	eMBReadInputStatus:
		MBV_Master.ReadInputStatus(
			Quantity								:= wMBVQuantity, 
			MBAddr									:= wMBVAddress, 
			cbLength								:= SIZEOF(wMBVReadData), 
			pMemoryAddr								:= ADR(wMBVReadData), 
			Execute									:= TRUE, 
			Timeout									:= MODBUS_TIMEOUT, 
			BUSY									=> bMBVBusy, 
			Error									=> bMBVError, 
			ErrorId									=> MBV_Errors, 
			cbRead									=> uiMBVRead);
		MBV_Master.ReadInputStatus(BUSY=> bMBVBusy);
		IF NOT MBV_Master.BUSY THEN
			MBV_Master.Execute 						:= FALSE;
			MBV_Master.ReadInputStatus(BUSY=> bMBVBusy);
			IF MBV_Master.Error THEN
				MBV_Master.ReadInputStatus();
			ELSE
				iMBVFunction 						:= 0;			
			END_IF
		END_IF
	
	eMBReadInputRegs:
		MBV_Master.ReadInputRegs(
			Quantity								:= wMBVQuantity, 
			MBAddr									:= wMBVAddress, 
			cbLength								:= SIZEOF(wMBVReadData), 
			pMemoryAddr								:= ADR(wMBVReadData), 
			Execute									:= TRUE, 
			Timeout									:= MODBUS_TIMEOUT, 
			BUSY									=> bMBVBusy, 
			Error									=> bMBVError, 
			ErrorId									=> MBV_Errors, 
			cbRead									=> uiMBVRead);
		MBV_Master.ReadInputRegs(BUSY=> bMBVBusy);
		IF NOT MBV_Master.BUSY THEN
			MBV_Master.Execute 						:= FALSE;
			MBV_Master.ReadInputRegs(BUSY=> bMBVBusy);
			IF MBV_Master.Error THEN
				MBV_Master.ReadInputRegs();
			ELSE
				iMBVFunction 						:= 0;			
			END_IF
		END_IF
	
	eMBWriteSingleCoil:
		MBV_Master.WriteSingleCoil(
			Quantity								:= wMBVQuantity, 
			MBAddr									:= wMBVAddress, 
			cbLength								:= SIZEOF(wMBVWriteData), 
			pMemoryAddr								:= ADR(wMBVWriteData), 
			Execute									:= TRUE, 
			Timeout									:= MODBUS_TIMEOUT, 
			BUSY									=> bMBVBusy, 
			Error									=> bMBVError, 
			ErrorId									=> MBV_Errors, 
			cbRead									=> uiMBVRead);
		MBV_Master.WriteSingleCoil(BUSY=> bMBVBusy);
		IF NOT MBV_Master.BUSY THEN
			MBV_Master.Execute 						:= FALSE;
			MBV_Master.WriteSingleCoil(BUSY=> bMBVBusy);
			IF MBV_Master.Error THEN
				MBV_Master.WriteSingleCoil();
			ELSE
				iMBVFunction 						:= 0;			
			END_IF
		END_IF
	
	eMBWriteMultipleCoils:
		MBV_Master.WriteMultipleCoils(
			Quantity								:= wMBVQuantity, 
			MBAddr									:= wMBVAddress, 
			cbLength								:= SIZEOF(wMBVWriteData), 
			pMemoryAddr								:= ADR(wMBVWriteData), 
			Execute									:= TRUE, 
			Timeout									:= MODBUS_TIMEOUT, 
			BUSY									=> bMBVBusy, 
			Error									=> bMBVError, 
			ErrorId									=> MBV_Errors, 
			cbRead									=> uiMBVRead);
		MBV_Master.WriteMultipleCoils(BUSY=> bMBVBusy);
		IF NOT MBV_Master.BUSY THEN
			MBV_Master.Execute 						:= FALSE;
			MBV_Master.WriteMultipleCoils(BUSY=> bMBVBusy);
			IF MBV_Master.Error THEN
				MBV_Master.WriteMultipleCoils();
			ELSE
				iMBVFunction 						:= 0;			
			END_IF
		END_IF
	
	eMBWriteRegs:
		MBV_Master.WriteRegs(
			Quantity								:= wMBVQuantity, 
			MBAddr									:= wMBVAddress, 
			cbLength								:= SIZEOF(wMBVWriteData), 
			pMemoryAddr								:= ADR(wMBVWriteData), 
			Execute									:= TRUE, 
			Timeout									:= MODBUS_TIMEOUT, 
			BUSY									=> bMBVBusy, 
			Error									=> bMBVError, 
			ErrorId									=> MBV_Errors, 
			cbRead									=> uiMBVRead);
		MBV_Master.WriteRegs(BUSY=> bMBVBusy);
		IF NOT MBV_Master.BUSY THEN
			MBV_Master.Execute 						:= FALSE;
			MBV_Master.WriteRegs(BUSY=> bMBVBusy);
			IF MBV_Master.Error THEN
				MBV_Master.WriteRegs();
			ELSE
				iMBVFunction 						:= 0;			
			END_IF
		END_IF
	
	ELSE
		iMBVFunction 								:= 0;
	
END_CASE
END_ACTION

ACTION A_Status_List:
// Calvin - A_Status_List
// Rev 1.00 - April 23, 2023

strStatusLabel[0] 									:= 'Start Warm Up';
strStatusLabel[1] 									:= 'Warm Up running';
strStatusLabel[2]  									:= 'Start Reactor Reset';
strStatusLabel[3]  									:= 'System ready';
strStatusLabel[4]  									:= 'Evacuation running';
strStatusLabel[5]  									:= 'Steam Bypass running';
strStatusLabel[6]  									:= 'Repressurization running';
strStatusLabel[7]  									:= 'Desorption running';
strStatusLabel[8]  									:= 'Adsorption running';
strStatusLabel[9]  									:= '';
strStatusLabel[10]  								:= 'Stopping process';
strStatusLabel[11]  								:= 'Stopping Warm Up';
strStatusLabel[12]  								:= 'Stopping Evacuation';
strStatusLabel[13]  								:= 'Stopping Steam Bypass';
strStatusLabel[14]  								:= 'Stopping Repressurization';
strStatusLabel[15]  								:= 'Stopping Desorption';
strStatusLabel[16]  								:= 'Stopping Adsorption';
strStatusLabel[17]  								:= '';
strStatusLabel[18]  								:= 'Cycle Error';
strStatusLabel[19]  								:= '';
strStatusLabel[20]  								:= '';
strStatusLabel[21]  								:= 'Fan Test Running';
strStatusLabel[22]  								:= 'Evacuation Error!';
strStatusLabel[23]  								:= 'Steam Bypass Error!';
strStatusLabel[24]  								:= 'Repressurization Error!';
strStatusLabel[25]  								:= 'Desorption Error!';
strStatusLabel[26]  								:= 'Adsorption Error!';
strStatusLabel[27]  								:= '';
strStatusLabel[28]  								:= '';
strStatusLabel[29]  								:= '';
strStatusLabel[30]  								:= 'Evacuation Complete';
strStatusLabel[31]  								:= 'Steam Bypass Complete';
strStatusLabel[32]  								:= 'Repressurization Complete';
strStatusLabel[33]  								:= 'Desoprtion Complete';
strStatusLabel[34]  								:= 'Adsorption Complete';
	
bStatusListLoaded									:= true;
END_ACTION

ACTION A_Temperatures:
// Calvin - A_Temperatures
// Rev 1.00 - June 26, 2023

tgr_TI_1001											:= F_Temperature(TI_1001);
tgb_TI_1001_Error									:= TI_1001_Error;
//bTI_1001_ErrActive									:= SEL(TI_1001_Error, FALSE, bTI_1001_ErrActive);
//gbAlarms[eTC_Alarm]									:= SEL(TI_1001_Error, gbAlarms[eTC_Alarm], TRUE);
                                    				
tgr_TI_1100A										:= F_Temperature(TI_1100A);
tgb_TI_1100A_Error									:= TI_1100A_Error;
//bTI_1100A_ErrActive									:= SEL(TI_1100A_Error, FALSE, bTI_1100A_ErrActive);
//gbAlarms[eTC_Alarm]									:= SEL(TI_1100A_Error, gbAlarms[eTC_Alarm], TRUE);
                                    				
tgr_TI_1100B										:= F_Temperature(TI_1100B);
tgb_TI_1100B_Error									:= TI_1100B_Error;
//bTI_1100B_ErrActive									:= SEL(TI_1100B_Error, FALSE, bTI_1100B_ErrActive);
//gbAlarms[eTC_Alarm]									:= SEL(TI_1100B_Error, gbAlarms[eTC_Alarm], TRUE);

tgr_TI_1100C										:= F_Temperature(TI_1100C);
tgb_TI_1100C_Error									:= TI_1100C_Error;
//bTI_1100C_ErrActive									:= SEL(TI_1100C_Error, FALSE, bTI_1100C_ErrActive);
//gbAlarms[eTC_Alarm]									:= SEL(TI_1100C_Error, gbAlarms[eTC_Alarm], TRUE);
                                    				
tgr_TI_1101											:= F_Temperature(TI_1101);
tgb_TI_1101_Error									:= TI_1101_Error;
//bTI_1101_ErrActive									:= SEL(TI_1101_Error, FALSE, bTI_1101_ErrActive);
//gbAlarms[eTC_Alarm]									:= SEL(TI_1101_Error, gbAlarms[eTC_Alarm], TRUE);
                                    				
tgr_TI_1102A										:= F_Temperature(TI_1102A);
tgb_TI_1102A_Error									:= TI_1102A_Error;
//bTI_1102A_ErrActive									:= SEL(TI_1102A_Error, FALSE, bTI_1102A_ErrActive);
//gbAlarms[eTC_Alarm]									:= SEL(TI_1102A_Error, gbAlarms[eTC_Alarm], TRUE);
                                    				
tgr_TI_1102B										:= F_Temperature(TI_1102B);
tgb_TI_1102B_Error									:= TI_1102B_Error;
//bTI_1102B_ErrActive									:= SEL(TI_1102B_Error, FALSE, bTI_1102B_ErrActive);
//gbAlarms[eTC_Alarm]									:= SEL(TI_1102B_Error, gbAlarms[eTC_Alarm], TRUE);
                                    				
tgr_TI_1103											:= F_Temperature(TI_1103);
tgb_TI_1103_Error									:= TI_1103_Error;
//bTI_1103_ErrActive									:= SEL(TI_1103_Error, FALSE, bTI_1103_ErrActive);
//gbAlarms[eTC_Alarm]									:= SEL(TI_1103_Error, gbAlarms[eTC_Alarm], TRUE);
                                    				
tgr_TI_1104											:= F_Temperature(TI_1104);
tgb_TI_1104_Error									:= TI_1104_Error;
//bTI_1104_ErrActive									:= SEL(TI_1104_Error, FALSE, bTI_1104_ErrActive);
//gbAlarms[eTC_Alarm]									:= SEL(TI_1104_Error, gbAlarms[eTC_Alarm], TRUE);
                                    				
tgr_TI_1105											:= F_Temperature(TI_1105);
tgb_TI_1105_Error									:= TI_1105_Error;
//bTI_1105_ErrActive									:= SEL(TI_1105_Error, FALSE, bTI_1105_ErrActive);
//gbAlarms[eTC_Alarm]									:= SEL(TI_1105_Error, gbAlarms[eTC_Alarm], TRUE);
                                    				
tgr_TI_1106											:= F_Temperature(TI_1106);
tgb_TI_1106_Error									:= TI_1106_Error;
//bTI_1106_ErrActive									:= SEL(TI_1106_Error, FALSE, bTI_1106_ErrActive);
//gbAlarms[eTC_Alarm]									:= SEL(TI_1106_Error, gbAlarms[eTC_Alarm], TRUE);
                                    				
tgr_TI_1301											:= F_Temperature(TI_1301);
tgb_TI_1301_Error									:= TI_1301_Error;
//bTI_1301_ErrActive									:= SEL(TI_1301_Error, FALSE, bTI_1301_ErrActive);
//gbAlarms[eTC_Alarm]									:= SEL(TI_1301_Error, gbAlarms[eTC_Alarm], TRUE);

tgr_TI_1302											:= F_Temperature(TI_1302);
tgb_TI_1302_Error									:= TI_1302_Error;
//bTI_1302_ErrActive									:= SEL(TI_1302_Error, FALSE, bTI_1302_ErrActive);
//gbAlarms[eTC_Alarm]									:= SEL(TI_1302_Error, gbAlarms[eTC_Alarm], TRUE);
                                    	
tgr_TI_1303											:= F_Temperature(TI_1303);
tgb_TI_1303_Error									:= TI_1303_Error;
//bTI_1303_ErrActive									:= SEL(TI_1303_Error, FALSE, bTI_1303_ErrActive);
//gbAlarms[eTC_Alarm]									:= SEL(TI_1303_Error, gbAlarms[eTC_Alarm], TRUE);
                                    				
tgr_TI_1304											:= F_Temperature(TI_1304);
tgb_TI_1304_Error									:= TI_1304_Error;
//bTI_1304_ErrActive									:= SEL(TI_1304_Error, FALSE, bTI_1304_ErrActive);
//gbAlarms[eTC_Alarm]									:= SEL(TI_1304_Error, gbAlarms[eTC_Alarm], TRUE);
                                    	
tgr_TI_1											:= F_Temperature(TI_1);
tgb_TI_1_Error										:= TI_1_Error;

tgr_TI_2											:= F_Temperature(TI_2);
tgb_TI_2_Error										:= TI_2_Error;

tgr_TI_3											:= F_Temperature(TI_3);
tgb_TI_3_Error										:= TI_3_Error;

tgr_TI_4											:= F_Temperature(TI_4);
tgb_TI_4_Error										:= TI_4_Error;

tgr_TI_5											:= F_Temperature(TI_5);
tgb_TI_5_Error										:= TI_5_Error;

tgr_TI_6											:= F_Temperature(TI_6);
tgb_TI_6_Error										:= TI_6_Error;

tgr_TI_7											:= F_Temperature(TI_7);
tgb_TI_7_Error										:= TI_7_Error;

tgr_TI_8											:= F_Temperature(TI_8);
tgb_TI_8_Error										:= TI_8_Error;

tgr_TI_9											:= F_Temperature(TI_9);
tgb_TI_9_Error										:= TI_9_Error;

tgr_TI_10											:= F_Temperature(TI_10);
tgb_TI_10_Error										:= TI_10_Error;

tgr_TI_11											:= F_Temperature(TI_11);
tgb_TI_11_Error										:= TI_11_Error;

tgr_TI_12											:= F_Temperature(TI_12);
tgb_TI_12_Error										:= TI_12_Error;

(*
IF gbAlarms[eTC_Alarm] AND NOT tgb_Active_Alarm THEN
	IF TI_1001_Error AND NOT bTI_1001_ErrActive AND giActiveAlarm = 0 THEN
		bTI_1001_ErrActive							:= TRUE;
		gsTempAlarm									:= '/ TI_1001';
		giActiveAlarm								:= eTC_Alarm;
	ELSIF TI_1100A_Error AND NOT bTI_1100A_ErrActive AND giActiveAlarm = 0 THEN
		bTI_1100A_ErrActive							:= TRUE;
		gsTempAlarm									:= '/ TI_1100A';
		giActiveAlarm								:= eTC_Alarm;
	ELSIF TI_1100B_Error AND NOT bTI_1100B_ErrActive AND giActiveAlarm = 0 THEN
		bTI_1100B_ErrActive							:= TRUE;
		gsTempAlarm									:= '/ TI_1100B';
		giActiveAlarm								:= eTC_Alarm;
	ELSIF TI_1100C_Error AND NOT bTI_1100C_ErrActive AND giActiveAlarm = 0 THEN
		bTI_1100C_ErrActive							:= TRUE;
		gsTempAlarm									:= '/ TI_1100C';
		giActiveAlarm								:= eTC_Alarm;
	ELSIF TI_1101_Error AND NOT bTI_1101_ErrActive AND giActiveAlarm = 0 THEN
		bTI_1101_ErrActive							:= TRUE;
		gsTempAlarm									:= '/ TI_1101';
		giActiveAlarm								:= eTC_Alarm;
	ELSIF TI_1102A_Error AND NOT bTI_1102A_ErrActive AND giActiveAlarm = 0 THEN
		bTI_1102A_ErrActive							:= TRUE;
		gsTempAlarm									:= '/ TI_1102A';
		giActiveAlarm								:= eTC_Alarm;
	ELSIF TI_1102B_Error AND NOT bTI_1102B_ErrActive AND giActiveAlarm = 0 THEN
		bTI_1102B_ErrActive							:= TRUE;
		gsTempAlarm									:= '/ TI_1102B';
		giActiveAlarm								:= eTC_Alarm;
	ELSIF TI_1103_Error AND NOT bTI_1103_ErrActive AND giActiveAlarm = 0 THEN
		bTI_1103_ErrActive							:= TRUE;
		gsTempAlarm									:= '/ TI_1103';
		giActiveAlarm								:= eTC_Alarm;
	ELSIF TI_1104_Error AND NOT bTI_1104_ErrActive AND giActiveAlarm = 0 THEN
		bTI_1104_ErrActive							:= TRUE;
		gsTempAlarm									:= '/ TI_1104';
		giActiveAlarm								:= eTC_Alarm;
	ELSIF TI_1105_Error AND NOT bTI_1105_ErrActive AND giActiveAlarm = 0 THEN
		bTI_1105_ErrActive							:= TRUE;
		gsTempAlarm									:= '/ TI_1105';
		giActiveAlarm								:= eTC_Alarm;
	ELSIF TI_1106_Error AND NOT bTI_1106_ErrActive AND giActiveAlarm = 0 THEN
		bTI_1106_ErrActive							:= TRUE;
		gsTempAlarm									:= '/ TI_1106';
		giActiveAlarm								:= eTC_Alarm;
	ELSIF TI_1301_Error AND NOT bTI_1301_ErrActive AND giActiveAlarm = 0 THEN
		bTI_1301_ErrActive							:= TRUE;
		gsTempAlarm									:= '/ TI_1301';
		giActiveAlarm								:= eTC_Alarm;
	ELSIF TI_1302_Error AND NOT bTI_1302_ErrActive AND giActiveAlarm = 0 THEN
		bTI_1302_ErrActive							:= TRUE;
		gsTempAlarm									:= '/ TI_1302';
		giActiveAlarm								:= eTC_Alarm;
	ELSIF TI_1303_Error AND NOT bTI_1303_ErrActive AND giActiveAlarm = 0 THEN
		bTI_1303_ErrActive							:= TRUE;
		gsTempAlarm									:= '/ TI_1303';
		giActiveAlarm								:= eTC_Alarm;
	ELSIF TI_1304_Error AND NOT bTI_1304_ErrActive AND giActiveAlarm = 0 THEN
		bTI_1304_ErrActive							:= TRUE;
		gsTempAlarm									:= '/ TI_1304';
		giActiveAlarm								:= eTC_Alarm;
	END_IF
END_IF
*)
END_ACTION

ACTION A_WaterHandling:
// Calvin - A_WaterHandling
// Rev 1.00 - September 21, 2023

IF bDrainOn OR tgb_Drains_On THEN
	
	tgb_HS_1200										:= NOT b1200DrainOROff;		//*** Interlock with error
	
	IF tgb_HS_1201_LSH OR (bClearDrains AND tgb_HS_1201_LSL) THEN															// 7/14/23 PS - Adsorption process change
		b1201DrainOn								:= TRUE;
	END_IF
	IF NOT tgb_HS_1201_LSL THEN
		b1201DrainOn								:= FALSE;
	END_IF
	tgb_HS_1201										:= b1201DrainOn AND (tgb_Drains_On OR NOT b1201DrainOROff);

	IF tgb_HS_1202_LSH OR (bClearDrains AND tgb_HS_1202_LSL) THEN															// 7/14/23 PS - Adsorption process change
		b1202DrainOn								:= TRUE;
	END_IF
	IF NOT tgb_HS_1202_LSL THEN
		b1202DrainOn								:= FALSE;
	END_IF
	tgb_HS_1202										:= b1300DrainOn OR b1202DrainOROn OR b1202DrainOn AND (tgb_Drains_On OR NOT b1202DrainOROff);
	tgb_HS_1300B									:= b1300DrainOn;
	
END_IF

rtrigDrainsOff(CLK:= NOT bDrainOn AND NOT tgb_Drains_On);																	// 09/20/23 PS
IF rtrigDrainsOff.Q THEN																									// 09/20/23 PS
	tgb_HS_1200										:= FALSE;
	tgb_HS_1201										:= FALSE;
	tgb_HS_1202										:= FALSE;
	tgb_HS_1300B									:= FALSE;
END_IF

bDrainLSHClear										:= NOT tgb_HS_1202_LSH AND NOT tgb_HS_1201_LSH;
bDrainLSLClear										:= NOT tgb_HS_1202_LSL AND NOT tgb_HS_1201_LSL; 

bCondenserLow										:= tgr_LI_1204 < CONDENSER_LEVEL_LOW_LIMIT;								// 09/19/23 PS
bCondenserFull										:= tgr_LI_1204 > CONDENSER_LEVEL_HIGH_LIMIT;							// 09/21/23 PS
bCondenserRefill									:= tgr_LI_1204 < CONDENSER_LEVEL_REFILL AND NOT bCondenserLow;			// 09/21/23 PS
END_ACTION

ACTION A0_Reset:
// Calvin - A0_Reset
// Rev 1.00 - September 21, 2023

tgr_HS_1102											:= 0;
tgr_IP_1102A										:= 0;
tgr_IP_1102B										:= 0;
tgr_IP_1101											:= 0;
tgr_IP_1302B										:= 0;
tgb_YL_1001											:= FALSE;
tgb_HS_1107											:= FALSE;				
tgb_HS_1101A										:= FALSE;
tgb_HS_1101B										:= FALSE;
tgb_AI_1102A_Pump									:= FALSE;
tgb_AI_1102A_Solenoid								:= FALSE;													
tgb_AI_1102B_Pump									:= FALSE;
tgb_AI_1102B_Solenoid								:= FALSE;													
tgb_HS_1103A										:= FALSE;				
tgb_HS_1103B										:= FALSE;				
tgb_HS_1104											:= FALSE;				
tgb_HS_1203											:= FALSE;				
tgb_HS_1302A										:= FALSE;				
tgb_HS_1301A										:= FALSE;				
tgb_HS_1301											:= FALSE;				
tgb_HS_1301B										:= FALSE;			
tgb_HS_1300A										:= FALSE;			
tgb_HS_1300B										:= FALSE;				
tgb_HS_1305											:= FALSE;
tgb_SV_1201											:= FALSE;
tgb_HT_1_On											:= FALSE;
tgb_HT_2_On											:= FALSE;
tgb_HT_3_On											:= FALSE;
tgb_HT_4_On											:= FALSE;
tgb_HT_5_On											:= FALSE;
tgb_HT_6_On											:= FALSE;
b1201DrainOROff										:= FALSE;
b1202DrainOROff										:= FALSE;
b1202DrainOROn										:= FALSE;
b1300DrainOn										:= FALSE;
bRunValveModulation									:= FALSE;
tgi_Current_Step									:= 0;
strProcessError										:= '';
END_ACTION

ACTION A1_WarmUp:
// Calvin - A1_WarmUp
// Rev 1.00 - September 22, 2023

CASE i1Step OF

	0:	;
	
	1:	
		A0_Reset();
		tgb_AI_1102A_Pump							:= TRUE;
		tgb_AI_1102B_Pump							:= TRUE;
		rTime1										:= VACUUM_TANK_DRAIN_TIME * SECONDS;
		strError									:= gsTK1300HighLevel;
		i1Step										:= i1Step + 1;

	2:	
		bTimer1										:= TRUE;
		IF tgb_HS_1300A_LSH THEN
			b1300DrainOn							:= TRUE;
		ELSE
			bTimer1									:= FALSE;
			b1300DrainOn							:= FALSE;
			IF bCondenserRefill THEN
				rTime2								:= 20 * SECONDS;
				tgb_SV_1201							:= TRUE;
				i1Step								:= i1Step + 1;
			ELSE
				rTime1								:= 10 * MINUTES;
				strError							:= gsBoilerPressureLow;
				i1Step								:= i1Step + 2;
			END_IF
		END_IF
		
	3:
		bTimer2										:= TRUE;
		IF tonTimer2.Q OR bCondenserFull THEN
			bTimer2									:= FALSE;
			tgb_SV_1201								:= FALSE;		
			rTime1									:= 10 * MINUTES;
			strError								:= gsBoilerPressureLow;
			i1Step									:= i1Step + 1;
		END_IF

	4:	
		bTimer1										:= TRUE;
		tgb_YL_1001									:= TRUE;
		IF tgr_PI_1001 > tgr_SP_Boiler_Pressure THEN
			bTimer1									:= FALSE;
			tgb_YL_1001								:= FALSE;
			tgb_Warmup_Complete						:= TRUE;
			i1Step									:= i1Step + 1;
		END_IF

	5:	
		bWarmUpDone									:= TRUE;
		tgi_Current_Step							:= 0;
		i1Step										:= 0;
	
END_CASE

strProcessError										:= SEL(bCondenserLow, strProcessError, gsLowCondenserLevel);					// 09/21/23 PS

IF i1Step > 0 THEN
	IF tonTimer1.Q OR tgb_Stop_Cycle OR strProcessError <> '' THEN
		giActiveAlarm 								:= SEL(tgb_Stop_Cycle, eWarmup_Alarm, eNo_Alarms);
		strError									:= SEL(strProcessError <> '', strError, strProcessError);
		iStep										:= i1Step;		
		A_ClearProcess();
		A0_Reset();
		i1Step										:= 5;
	END_IF
	tgi_Current_Step								:= i1Step;
END_IF
END_ACTION

ACTION A2_Evacuation:
// Calvin - A2_Evacuation
// Rev 1.00 -September 22, 2023

CASE i2Step OF
	
	0:	;
	
	1:	
		A0_Reset();
		tgb_AI_1102A_Pump							:= TRUE;
		tgb_AI_1102B_Pump							:= TRUE;
		gbVacuumHolding								:= FALSE;
		rTime1										:= 30 * SECONDS;
		i2Step										:= 2;
				
	2:	
		IF bDrainLSHClear THEN
			strError								:= gsValvesNotClosed;
			i2Step									:= 4;
		ELSE
			strError								:= gsDrainNotClear;
			i2Step									:= i2Step + 1;
		END_IF
	
	3:	
		bTimer1										:= TRUE;
		IF bDrainLSHClear AND bDrainLSLClear THEN
			bTimer1									:= FALSE;
			strError								:= gsValvesNotClosed;
			i2Step									:= i2Step + 1;
		END_IF

	4:	
		bTimer1										:= TRUE;
		IF gbHS_1102ValvesClosed THEN
			bTimer1									:= FALSE;
			rTime1									:= DEFAULT_STEP_TIME;
			strError								:= gsLRPCoolingFlowLow;
			i2Step									:= i2Step + 1;
		END_IF
	
	5:	
		bTimer1										:= TRUE;
		IF tgb_HS_1300A_LSL AND NOT tgb_HS_1300A_LSH THEN
			tgb_HS_1300A							:= TRUE;
			tgb_HS_1305								:= TRUE;
			tgb_HS_1301								:= TRUE;			
			bTimer1									:= FALSE;
			rTime2									:= 5 * SECONDS;
			i2Step									:= i2Step + 1;
		END_IF
		
	6:	
		bTimer2										:= TRUE;
		IF tonTimer2.Q THEN
			bTimer2									:= FALSE;
			rTime1									:= DEFAULT_STEP_TIME;
			rSP1									:= tgr_SP_Min_LRP_Cooling_Loop_Flow;
			strError								:= gsLRPCoolingFlowLow;
			i2Step									:= i2Step + 1;
		END_IF
	
	7:	
		bTimer1										:= TRUE;
		IF tgr_FI_1300 > rSP1 THEN
			bTimer1									:= FALSE;
			rTime1									:= DEFAULT_STEP_TIME;
			strError								:= gsDrainNotClear;
			i2Step									:= i2Step + 1;
		END_IF			

	8:	
		bTimer1										:= TRUE;
		IF bDrainLSHClear THEN
			b1201DrainOROff							:= TRUE;
			b1202DrainOROff							:= TRUE;
			bTimer1									:= FALSE;
			rTime1									:= DEFAULT_STEP_TIME;
			rSP1									:= tgr_SP_Evacuation_Target_Pressure;
			strError								:= gsTargetPressureHigh;
			i2Step									:= i2Step + 1;
		END_IF
		
	9:	
		bTimer1										:= TRUE;
		IF tgr_PI_1300 < rSP1 THEN
			tgb_HS_1302A							:= TRUE;
			tgb_HS_1107								:= TRUE;
			bTimer1									:= FALSE;
			rTime2									:= 10 * SECONDS;
			i2Step									:= i2Step + 1;
		END_IF

	10:	
		bTimer2										:= TRUE;
		IF tonTimer2.Q THEN
			bTimer2									:= FALSE;
			rTime1									:= DEFAULT_STEP_TIME;
			rSP1									:= tgr_SP_Evacuation_Target_Pressure;
			strError								:= gsTargetPressureHigh;
			i2Step									:= i2Step + 1;
		END_IF
	
	11:	
		bTimer1										:= TRUE;
		IF tgr_PI_1300 <= rSP1 THEN
			bTimer1									:= FALSE;
			tgb_HS_1103A							:= TRUE;
			tgb_HS_1103B							:= TRUE;
			rTime2									:= 10 * SECONDS;
			i2Step									:= i2Step + 1;
		END_IF
		
	12:	
		bTimer2										:= TRUE;
		IF tonTimer2.Q THEN
			bTimer2									:= FALSE;
			rTime1									:= 5 * MINUTES;
			rSP1									:= tgr_SP_Evacuation_Target_Pressure;
			i2Step									:= i2Step + 1;
		END_IF
	
   	13:	
		bTimer1										:= TRUE;
		bInRange1									:= tgr_PI_1300 < rSP1;
		bInRange2									:= tgr_PI_1100 <= rSP1;
		strError									:= SEL(bInRange1, gsPI_1300OutOfRange, gsPI_1100OutOfRange);
		IF bInRange1 AND bInRange2 THEN
			bTimer1									:= FALSE;
			tgb_HS_1103A							:= FALSE;
 	  		tgb_HS_1103B							:= FALSE;
			tgb_HS_1302A							:= FALSE;
			tgb_HS_1301								:= FALSE;
			tgb_HS_1300A							:= FALSE;
			tgb_HS_1305								:= FALSE;
			tgb_HS_1107								:= FALSE;
			rPI_1100_Save							:= tgr_PI_1100;
			rTime2									:= tgr_SP_Leak_Check_Time * SECONDS;
			i2Step									:= i2Step + 1;
		END_IF

	14:	
		bTimer2										:= TRUE;
		IF tonTimer2.Q THEN
			bTimer2									:= FALSE;
			rTime1									:= SECONDS;
			rSP1									:= tgr_SP_Max_Allowed_Pressure_Leakage;
			strError								:= gsVacuumLeak;
			i2Step									:= i2Step + 1;
		END_IF
	
	15:	
		bTimer1										:= TRUE;
		IF ABS(tgr_PI_1100 - rPI_1100_Save) <= rSP1 THEN
			bTimer1									:= FALSE;
			gbVacuumHolding							:= TRUE;
			i2Step									:= i2Step + 1;
		END_IF

	16:	
		b1201DrainOROff								:= FALSE;
		b1202DrainOROff								:= FALSE;
		bEvacuationDone								:= TRUE;
		tgi_Current_Step							:= 0;
		i2Step										:= 0;
		
END_CASE
		
IF i2Step > 0 THEN
	IF tonTimer1.Q OR tgb_Stop_Cycle OR strProcessError <> '' THEN
		giActiveAlarm 								:= SEL(tgb_Stop_Cycle, eEvacuation_Alarm, eNo_Alarms);
		strError									:= SEL(strProcessError <> '', strError, strProcessError);
		iStep										:= i2Step;		
		A_ClearProcess();
		A0_Reset();
		i2Step										:= 16;
	END_IF
	tgi_Current_Step								:= i2Step;
END_IF
END_ACTION

ACTION A3_SteamBypass:
// Calvin - A3_SteamBypass
// Rev 1.00 - September 22, 2023

CASE i3Step OF
	
	0:	;

	1:	
		A0_Reset();
		tgb_AI_1102A_Pump							:= TRUE;
		tgb_AI_1102B_Pump							:= TRUE;
		YL_1001										:= TRUE;
		rTime1										:= VACUUM_TANK_DRAIN_TIME * SECONDS;
		strError									:= gsTK1300HighLevel;
		i3Step										:= i3Step + 1;

	2:	
		bTimer1										:= TRUE;
		IF tgb_HS_1300A_LSH THEN
			b1300DrainOn							:= TRUE;
		ELSE
			bTimer1									:= FALSE;
			b1300DrainOn							:= FALSE;
			IF bCondenserRefill THEN
				rTime2								:= 20 * SECONDS;
				i3Step								:= i3Step + 1;
			ELSE
				rTime1								:= 3 * MINUTES;
				strError							:= gsBoilerPressureLow;
				i3Step								:= i3Step + 2;
			END_IF
		END_IF
		
	3:
		bTimer1										:= TRUE;
		IF NOT bCondenserRefill OR bCondenserFull THEN
			bTimer1									:= FALSE;
			tgb_SV_1201								:= FALSE;		
			tgb_YL_1001								:= TRUE;
			b1201DrainOROff							:= TRUE;
			rTime1									:= 3 * MINUTES;
			i3Step									:= i3Step + 1;
		ELSE
			tgb_SV_1201								:= TRUE;
		END_IF
		
	4:	
		bTimer1										:= TRUE;
		strError									:= SEL(tgr_PI_1101 >= tgr_SP_Evacuation_Target_Pressure_Steam, gsBoilerPressureLow, gsTargetPressureHigh);
		IF tgr_PI_1101 < tgr_SP_Evacuation_Target_Pressure_Steam AND tgr_PI_1001 >= tgr_SP_Boiler_Pressure THEN
			bTimer1									:= FALSE;
			b1202DrainOROn							:= TRUE;
			tgb_HS_1203								:= TRUE;
			tgr_IP_1101								:= 100;
			tgb_HS_1107								:= TRUE;
			rTime2									:= 60 * SECONDS;
			i3Step									:= i3Step + 1;
		END_IF
	
	5:	
		bTimer2										:= TRUE;
		IF tonTimer2.Q THEN
			bTimer2									:= FALSE;
			rTime1									:= 3 * MINUTES;
			strError								:= gsSteamFlowLow;
			i3Step									:= i3Step + 1;
		END_IF
		
	6:	
		bTimer1										:= TRUE;
		IF tgr_FI_1001 > tgr_SP_Min_Bypass_Steam_Flow THEN
			bTimer1									:= FALSE;
			rTime2									:= 30 * SECONDS;
			i3Step									:= i3Step + 1;
		END_IF
		
	7:	
		bTimer2										:= TRUE;
		IF tonTimer2.Q THEN
			bTimer2									:= FALSE;
			rTime1									:= 5 * MINUTES;
			strError								:= gsSteamTempLow;
			i3Step									:= i3Step + 1;
		END_IF
	
	8:	
		bTimer1										:= TRUE;
		strProcessError								:= SEL(tgb_TI_1101_Error, strProcessError, gsTI_1101Error);					// 09/20/23 PS
		IF tgr_TI_1101 > tgr_SP_Min_Bypass_Steam_Temp THEN
			bTimer1									:= FALSE;
			tgr_IP_1101								:= 0;
			tgb_HS_1107								:= FALSE;
			rTime1									:= 10 * MINUTES;
			strError								:= gsLimitSwitchError;
			i3Step									:= i3Step + 1;
		END_IF
		
	9:	
		bTimer1										:= TRUE;
		IF NOT tgb_HS_1202_LSH THEN
			bTimer1									:= FALSE;
			b1202DrainOROff							:= TRUE;
			b1202DrainOROn							:= FALSE;
			tgb_HS_1203								:= FALSE;
			i3Step									:= i3Step + 1;
		END_IF
		
	10:	
		bSteamBypassDone							:= TRUE;
		tgi_Current_Step							:= 0;
		i3Step										:= 0;
		
END_CASE
		
strProcessError										:= SEL(bCondenserLow, strProcessError, gsLowCondenserLevel);					// 09/20/23 PS

IF i3Step > 0 THEN
	IF tonTimer1.Q OR tgb_Stop_Cycle OR strProcessError <> '' THEN
		giActiveAlarm 								:= SEL(tgb_Stop_Cycle, eSteamBypass_Alarm, eNo_Alarms);
		strError									:= SEL(strProcessError <> '', strError, strProcessError);		
		iStep										:= i3Step;		
		A_ClearProcess();
		A0_Reset();
		i3Step										:= 10;
	END_IF
	tgi_Current_Step								:= i3Step;
END_IF
END_ACTION

ACTION A4_Desorption:
// Calvin - A4_Desorption
// Rev 1.00 - September 22, 2023

CASE i4Step OF
	
	0:	bOverTemp									:= FALSE;
		
	1:	
		A0_Reset();
		YL_1001										:= TRUE;
		b1201DrainOROff								:= TRUE;
		b1202DrainOROff								:= TRUE;
		rTime1										:= 2 * SECONDS;
		rSP1										:= tgr_SP_Evacuation_Target_Pressure_Steam;								// 07/14/23 PS - Added set point
		strError									:= gsTargetPressureHigh;
		i4Step										:= 2;
	
	2:	
		bTimer1										:= TRUE;
		IF tgr_PI_1100 < rSP1 THEN
			bTimer1									:= FALSE;
			i4Step									:= i4Step + 1;
		END_IF
		
	3:	
		IF gbVacuumHolding THEN
			rTime1									:= DEFAULT_STEP_TIME;
			rSP1									:= tgr_SP_Evacuation_Target_Pressure_Steam;								// 07/14/23 PS - Added set point
			rSP2									:= tgr_SP_Boiler_Pressure;
			i4Step									:= 6;
		ELSE
			rTime2									:= tgr_SP_Leak_Check_Time * SECONDS;
			i4Step									:= i4Step + 1;
		END_IF
		
	4:	
		bTimer2										:= TRUE;
		IF tonTimer2.Q THEN
			bTimer2									:= FALSE;
			rTime1									:= 1 * SECONDS;
			rSP1									:= tgr_SP_Max_Allowed_Pressure_Leakage;
			strError								:= gsVacuumLeak;
			i4Step									:= i4Step + 1;
		END_IF

	5:	
		bTimer1										:= TRUE;
		IF ABS(tgr_PI_1100 - rPI_1100_Save) <= rSP1 THEN
			bTimer1									:= FALSE;
			gbVacuumHolding							:= TRUE;
			rTime1									:= 10 * MINUTES;
			rSP1									:= tgr_SP_Evacuation_Target_Pressure_Steam;								// 07/14/23 PS - Added set point
			rSP2									:= tgr_SP_Boiler_Pressure;
			i4Step									:= i4Step + 1;
		END_IF

	6:	
		bTimer1										:= TRUE;
		bInRange1									:= tgr_PI_1100 < rSP1;
		bInRange2									:= tgr_PI_1001 >= rSP2;
		strError									:= SEL(bInRange1, gsTargetPressureHigh, gsBoilerPressureLow);
		IF bInRange1 AND bInRange2 THEN
			bTimer1									:= FALSE;
			rTime2									:= 5 * SECONDS;
			i4Step									:= i4Step + 1;
		END_IF
		
	7:	
		bTimer2										:= TRUE;
		tgr_IP_1101									:= tgr_SP_Steam_Valve_Percent_Open;
		IF tonTimer2.Q THEN
			bTimer2									:= FALSE;
			rTime1									:= DEFAULT_STEP_TIME;
			strError								:= gsValveOutOfRange;
			i4Step									:= i4Step + 1;
		END_IF
		
	8:	
		bTimer1										:= TRUE;
		bInRange1									:= ABS(tgr_ZT_1101 - tgr_IP_1101) <= 5;
 		IF bInRange1 THEN
			bTimer1									:= FALSE;
			tgb_HS_1101A							:= TRUE;
			tgb_HS_1101B							:= TRUE;
			rTime1									:= 10 * MINUTES;
			strError								:= gsReactorPressureLow;
			i4Step									:= i4Step + 1;
		END_IF

	9:	
		bTimer1										:= TRUE;
		IF tgr_PI_1100 > 0.5 THEN
			bTimer1									:= FALSE;
			gbVacuumHolding							:= FALSE;
			b1201DrainOROff							:= FALSE;
			b1202DrainOROff							:= FALSE;
			rTime1									:= 30 * MINUTES;
			rSP1									:= tgr_SP_Steam_Repressurization_Pressure;
			i4Step									:= i4Step + 1;
		END_IF

	10:	
		bTimer1										:= TRUE;	
		bInRange1									:= tgr_PI_1001 > rSP1;
		bInRange2									:= tgr_PI_1101 > rSP1;
		bInRange3									:= tgr_PI_1100 > rSP1;
		strError									:= SEL(bInRange1, gsPI_1001PressureLow, SEL(bInRange2, gsPI_1101PressureLow, gsPI_1100PressureLow));
		IF bInRange1 AND bInRange2 AND bInRange3 THEN
			bTimer1									:= FALSE;
			tgb_HS_1203								:= TRUE;
			tgb_HS_1300A							:= TRUE;
			tgb_HS_1305								:= TRUE;
			tgb_HS_1301								:= TRUE;
			rTime2									:= 5 * SECONDS;
			i4Step									:= i4Step + 1;
		END_IF
		
	11:	
		bTimer2										:= TRUE;
		IF tonTimer2.Q THEN
			bTimer2									:= FALSE;
			rTime1									:= 20 * SECONDS;
			rSP1									:= tgr_SP_Min_LRP_Cooling_Loop_Flow;
			rSP2									:= tgr_SP_Evacuation_Target_Pressure;
			i4Step									:= i4Step + 1;
		END_IF
	
	12:	
		bTimer1										:= TRUE;
		bInRange1									:= tgr_FI_1300 > rSP1;
		bInRange2									:= tgr_PI_1300 < rSP2;
		IF bInRange1 AND bInRange2 THEN
			bTimer1									:= FALSE;
			tgb_HS_1302A							:= TRUE;
			rTime2									:= 6 * SECONDS;
			i4Step									:= i4Step + 1;
		END_IF
		
	13:	
		bTimer2										:= TRUE;
		IF tonTimer2.Q THEN
			bTimer2									:= FALSE;
			rSP1									:= tgr_SP_Evacuation_Target_Pressure;
			i4Step									:= i4Step + 1;
		END_IF

	14:	
		IF tgr_PI_1300 < rSP1 THEN
			tgr_IP_1302B							:= tgr_SP_IP_1302B_Valve_Low;
		END_IF
		rTime2										:= 3 * SECONDS;
		i4Step										:= i4Step + 1;
		
	15:	
		bTimer2										:= TRUE;
		IF tonTimer2.Q THEN
			bTimer2									:= FALSE;
			rSP1									:= tgr_SP_Evacuation_Target_Pressure;
			strError								:= gsTargetPressureHigh;
			i4Step									:= i4Step + 1;
		END_IF

	16:	
		bTimer1										:= TRUE;
		IF tgr_PI_1300 < rSP1 THEN
			bTimer1									:= FALSE;
			tgb_HS_1103A							:= TRUE;
			tgb_HS_1103B							:= TRUE;
			bRunValveModulation						:= TRUE;
			rTime1									:= 5 * MINUTES;
			rTime2									:= tgr_SP_Steam_Purge_Time * MINUTES;
			strError								:= gsValveOutOfRange;
			i4Step									:= i4Step + 1;
		END_IF
		
	17:	
		bTimer1										:= TRUE;
		bTimer2										:= TRUE;
		IF bValveInRange THEN
			bTimer1									:= FALSE;
			rTime1									:= SECONDS;
			strError								:= gsThermocoupleError;
			i4Step									:= i4Step + 1;
		END_IF
		
	18:	
		bTimer1										:= TRUE;
		IF NOT tgb_TI_1100A_Error OR NOT tgb_TI_1100B_Error OR NOT tgb_TI_1100C_Error THEN
			bTimer1									:= FALSE;
			rSP1									:= tgr_SP_Max_Allowed_Sorbent_Temp;
			rSP2									:= tgr_SP_Steam_Purge_Cutoff_Temp;
			i4Step									:= i4Step + 1;
		END_IF
	
	19:	
		bInRange1									:= NOT tgb_TI_1100A_Error AND tgr_TI_1100A > rSP1;
		bInRange2									:= NOT tgb_TI_1100B_Error AND tgr_TI_1100B > rSP1;
		bInRange3									:= NOT tgb_TI_1100C_Error AND tgr_TI_1100C > rSP1;
		IF bInRange1 OR bInRange2 OR bInRange3 THEN
			bOverTemp								:= TRUE;
			bTimer2									:= FALSE;
			rTime1									:= SECONDS;
			i4Step									:= i4Step + 1;
		ELSE
			bInRange1								:= (NOT tgb_TI_1100A_Error AND tgr_TI_1100A > rSP2) OR tgb_TI_1100A_Error;
			bInRange2								:= (NOT tgb_TI_1100B_Error AND tgr_TI_1100B > rSP2) OR tgb_TI_1100B_Error;
			bInRange3								:= (NOT tgb_TI_1100C_Error AND tgr_TI_1100C > rSP2) OR tgb_TI_1100C_Error;
			IF tonTimer2.Q THEN
				bTimer2								:= FALSE;
				IF bInRange1 AND bInRange2 AND bInRange3 THEN
					i4Step							:= i4Step + 1;
				ELSE
					strProcessError					:= SEL(bOverTemp, gsTempOutOfRange, gsSorbentOverTemp);
				END_IF
			END_IF
		END_IF
		
	20:	
		bRunValveModulation							:= FALSE;
		tgr_IP_1101									:= 0;
		tgr_IP_1302B								:= 0;
		tgb_HS_1101A								:= FALSE;							
		tgb_HS_1101B								:= FALSE;							
		rTime1										:= 5 * MINUTES;
		rSP1										:= 0.5;
		strError									:= gsPI_1100OutOfRange;
		i4Step										:= i4Step + 1;	

	21: 
		bTimer1										:= TRUE;
		IF tgr_PI_1100 < rSP1 THEN
			bTimer1									:= FALSE;
			b1201DrainOROff							:= TRUE;
			b1202DrainOROff							:= TRUE;
			rSP1									:= tgr_SP_Evap_Cooling_Cutoff_Temp;
			rSP2									:= tgr_SP_Evap_Cooling_Target_Pressure;
			rTime1									:= 20 * MINUTES;
			i4Step									:= i4Step + 1;
		END_IF
		
	22:	
		bTimer1										:= TRUE;
		bInRange1									:= (NOT tgb_TI_1100A_Error AND tgr_TI_1100A < rSP1) OR tgb_TI_1100A_Error;
		bInRange2									:= (NOT tgb_TI_1100B_Error AND tgr_TI_1100B < rSP1) OR tgb_TI_1100B_Error;
		bInRange3									:= (NOT tgb_TI_1100C_Error AND tgr_TI_1100C < rSP1) OR tgb_TI_1100C_Error;
		strError									:= SEL(tgr_PI_1100 >= rSP2, gsTempOutOfRange, gsPI_1100OutOfRange);
		IF bInRange1 AND bInRange2 AND bInRange3 AND tgr_PI_1100 < rSP2 THEN
			bTimer1									:= FALSE;
			i4Step									:= i4Step + 1;
		END_IF	
		
	23:	
		tgb_HS_1103A								:= FALSE;
		tgb_HS_1103B								:= FALSE;
		tgb_HS_1302A								:= FALSE;
		tgb_HS_1301									:= FALSE;
		tgb_HS_1305									:= FALSE;
		tgb_HS_1300A								:= FALSE;
		tgb_HS_1203									:= FALSE;
		i4Step										:= i4Step + 1;
		
	24:
		bDesorptionDone								:= TRUE;
		tgi_Current_Step							:= 0;
		i4Step										:= 0;		
	
END_CASE

strProcessError										:= SEL(bCondenserLow, strProcessError, gsLowCondenserLevel);					// 09/07/23 PS

IF i4Step > 0 THEN
	IF tonTimer1.Q OR tgb_Stop_Cycle OR strProcessError <> '' THEN
		giActiveAlarm 								:= SEL(tgb_Stop_Cycle, eDesorption_Alarm, eNo_Alarms);
		strError									:= SEL(strProcessError <> '', strError, strProcessError);		
		iStep										:= i4Step;		
		A_ClearProcess();
		A0_Reset();
		i4Step										:= 24;
	END_IF
	tgi_Current_Step								:= i4Step;
END_IF
END_ACTION

ACTION A5_Repressurization:
// Calvin - A5_Repressurization
// Rev 1.00 - September 22, 2023

CASE i5Step OF
	
	0:	;
		
	1:	
		A0_Reset();
		tgb_AI_1102A_Pump							:= TRUE;
		tgb_AI_1102B_Pump							:= TRUE;
		rTime1										:= SECONDS;
		strError									:= gsThermocoupleError;
		i5Step										:= 2;
		
	2:	
		bTimer1										:= TRUE;
		bTempAGood									:= NOT tgb_TI_1100A_Error;
		bTempBGood									:= NOT tgb_TI_1100B_Error;
		bTempCGood									:= NOT tgb_TI_1100C_Error;
		IF bTempAGood OR bTempBGood OR bTempCGood THEN
			bTimer1									:= FALSE;
			rTime1									:= DEFAULT_STEP_TIME;
			rSP1									:= tgr_SP_Adsorption_Temp;
			strError								:= gsTempOutOfRange;
			i5Step									:= i5Step + 1;
		END_IF
	
	3:	
		bTimer1										:= TRUE;
		bInRange1									:= (bTempAGood AND tgr_TI_1100A < rSP1) OR NOT bTempAGood;
		bInRange2									:= (bTempBGood AND tgr_TI_1100B < rSP1) OR NOT bTempBGood;
		bInRange3									:= (bTempCGood AND tgr_TI_1100C < rSP1) OR NOT bTempCGood;
		IF bInRange1 AND bInRange2 AND bInRange3 THEN
			bTimer1									:= FALSE;
			tgb_HS_1104								:= TRUE;
			rTime1									:= DEFAULT_STEP_TIME;
			rSP1									:= tgr_SP_Reactor_Repressurization_Pressure;
			strError								:= gsPI_1100OutOfRange;			
			i5Step									:= i5Step + 1;
		END_IF
		
	4:	
		bTimer1										:= TRUE;
		IF tgr_PI_1100 > rSP1 THEN
			bTimer1									:= FALSE;
			rTime2									:= 5 * SECONDS;
			i5Step									:= i5Step + 1;			
		END_IF
		
	5:	
		bTimer2										:= TRUE;
		IF tonTimer2.Q THEN
			bTimer2									:= FALSE;
			i5Step									:= i5Step + 1;
		END_IF
		
	6:	
		tgb_HS_1104									:= FALSE;
		i5Step										:= i5Step + 1;
	
	7:	
		bRepressurizationDone						:= TRUE;
		tgi_Current_Step							:= 0;
		i5Step										:= 0;
	
END_CASE

IF i5Step > 0 THEN
	IF tonTimer1.Q OR tgb_Stop_Cycle OR strProcessError <> '' THEN
		giActiveAlarm 								:= SEL(tgb_Stop_Cycle, eRepressurization_Alarm, eNo_Alarms);
		strError									:= SEL(strProcessError <> '', strError, strProcessError);		
		iStep										:= i5Step;		
		A_ClearProcess();
		A0_Reset();
		i5Step										:= 7;
	END_IF
	tgi_Current_Step								:= i5Step;
END_IF
END_ACTION

ACTION A6_Adsorption:
// Calvin - A6_Adsorption
// Rev 1.00 - September 22, 2023

CASE i6Step OF
	
	0:	;
		
	1:	
		A0_Reset();
		tgb_AI_1102A_Pump							:= TRUE;
		tgb_AI_1102B_Pump							:= TRUE;
		bClearDrains								:= FALSE;
		rSP1										:= tgr_SP_Reactor_Repressurization_Pressure;
		strError									:= gsReactorPressureLow;
		rTime1										:= 5 * MINUTES;
		i6Step										:= i6Step + 1;
	
	2:	
		bTimer1										:= TRUE;
		IF tgr_PI_1100 > rSP1 THEN
			tgr_IP_1102A							:= 100;
			tgr_IP_1102B							:= 100;
			bTimer1									:= FALSE;
			rTime1									:= DEFAULT_STEP_TIME;
			strError								:= gsValvesNotOpen;
			i6Step									:= i6Step + 1;
		END_IF
		
	3:	
		bTimer1										:= TRUE;
		IF gbHS_1102ValvesOpen THEN																		// Valves are fully open
			bTimer1									:= FALSE;
			tgr_HS_1102								:= tgr_SP_Adsorption_VFD_Output;
			bFanError								:= tgb_Auto_Mode;									// Run evacuation if cycling
			rTime1									:= DEFAULT_STEP_TIME;
			rSP1									:= 20;
			strError								:= gsNoAirFlow;
			i6Step									:= i6Step + 1;
		END_IF
	
	4:	
		bTimer1										:= TRUE;
		IF tgr_FIC_1102 > rSP1 THEN																		// Verify fan operation with air flow
			bTimer1									:= FALSE;
			bFanError								:= FALSE;
			rTime2									:= 30 * SECONDS;
			i6Step									:= i6Step + 1;
		END_IF
	
	5:	
		bTimer2										:= TRUE;
		IF tonTimer2.Q THEN
			bTimer2									:= FALSE;
			rTime2									:= SEL(tgb_Adsorption_CO2, tgr_SP_Adsorption_Time, tgr_SP_Adsorption_CO2_Time) * MINUTES;
			rTime1									:= rTime2 + SECONDS;																			// Add extra second to allow Timer2 to time out first
			rSP1									:= tgr_SP_Adsorption_CO2_Differential;
			strError								:= gsCO2DifferentialError;
			i6Step									:= i6Step + 1;
		END_IF
		
	6:	
		bTimer1										:= TRUE;
		bTimer2										:= TRUE;
		bInRange1									:= SEL(tgb_Adsorption_CO2, tonTimer2.Q, ABS(tgr_AI_1102A - tgr_AI_1102B) < rSP1);
		i6Step										:= SEL(bInRange1, i6Step, i6Step + 1);
		
	7:	
		bTimer1										:= FALSE;
		bTimer2										:= FALSE; 
		tgr_HS_1102									:= 0;
		rTime1										:= DEFAULT_STEP_TIME;
		strError									:= gsFanStillRunning;
		i6Step										:= i6Step + 1;
		
	8:	
		bTimer1										:= TRUE;
		IF tgr_HS_1102_RPM = 0 THEN
			bTimer1									:= FALSE;
			tgb_AI_1102A_Pump						:= FALSE;
			tgb_AI_1102A_Solenoid					:= FALSE;													
			tgb_AI_1102B_Pump						:= FALSE;
			tgb_AI_1102B_Solenoid					:= FALSE;													
			bClearDrains							:= TRUE;
			rTime2									:= 5 * MINUTES;
			i6Step									:= i6Step + 1;
		END_IF

	9:	
		bTimer2										:= TRUE;
		IF tonTimer2.Q OR (NOT tgb_HS_1201_LSL AND NOT tgb_HS_1202_LSL) THEN
			bTimer2									:= FALSE;
			bClearDrains							:= FALSE;
			tgr_IP_1102A							:= 0;
			tgr_IP_1102B							:= 0;
			rTime1									:= DEFAULT_STEP_TIME;
			strError								:= gsValvesNotClosed;
			i6Step									:= i6Step + 1;
		END_IF

	10:	
		bTimer1										:= TRUE;
		IF gbHS_1102ValvesClosed THEN
			bTimer1									:= FALSE;
			i6Step									:= i6Step + 1;
		END_IF

	11:	
		bAdsorptionDone								:= TRUE;
		tgi_Current_Step							:= 0;
		i6Step										:= 0;

END_CASE

IF i6Step > 0 THEN
	IF tonTimer1.Q OR tgb_Stop_Cycle OR strProcessError <> '' THEN
		giActiveAlarm 								:= SEL(tgb_Stop_Cycle, eAdsorption_Alarm, eNo_Alarms);
		strError									:= SEL(strProcessError <> '', strError, strProcessError);		
		iStep										:= i6Step;		
		A_ClearProcess();
		A0_Reset();
		i6Step										:= 11;
	END_IF
	tgi_Current_Step								:= i6Step;
END_IF
END_ACTION

END_PROGRAM

// ---- POUs/Functions/F_AnalogIn.TcPOU
FUNCTION F_AnalogIn : REAL
VAR_INPUT
	Input											: INT;
	Low												: REAL;
	High											: REAL;
	Minimum											: REAL;
	Offset											: REAL;
END_VAR
VAR
	Value											: REAL;
END_VAR

// Calvin - F_AnalogIn
// Rev 1.0 - March 3, 2023

Value												:= ((High - Low) / 32767.0) * INT_TO_REAL(Input) + Low;		// Determine output based on scale
Value												:= Value + Offset;											// Adjust for any user offset
F_AnalogIn											:= SEL(ABS(Value) > Minimum, 0, Value);						// Value must be above (or below, if negative) minimum or zero is returned

END_FUNCTION

// ---- POUs/Functions/F_Current.TcPOU
FUNCTION F_Current : REAL
VAR_INPUT
	I_Reading				: INT;
END_VAR
VAR
END_VAR

// Calvin - F_Current
// Rev 1.0 - April 6, 2023

F_Current					:= INT_TO_REAL(I_Reading) / 163.835;

END_FUNCTION

// ---- POUs/Functions/F_Voltage.TcPOU
FUNCTION F_Voltage : REAL
VAR_INPUT
	V_Reading				: INT;
END_VAR
VAR
END_VAR

// Calvin - F_Voltage
// Rev 1.0 - April 6, 2023

F_Voltage					:= INT_TO_REAL(V_Reading) / 65.534;

END_FUNCTION

// ---- POUs/Functions/F_Temperature.TcPOU
FUNCTION F_Temperature : REAL
VAR_INPUT
	Input											: INT;
END_VAR
VAR
END_VAR

// Calvin - F_Temperature
// Rev 1.0 - March 3, 2023

F_Temperature										:= INT_TO_REAL(Input) / 10.0;

END_FUNCTION

// ---- POUs/P_AlarmCheck.TcPOU
PROGRAM P_AlarmCheck
VAR
	rtrigCheckErrors								: R_TRIG;
	ftrigClearError									: F_TRIG;
	tonAlarmTimer									: TON;
	i												: INT;
	iMultipleTempError								: INT;
	iErrorCount										: INT;
	iCount											: INT;
	iDisplayAlarm									: INT := 1;
	iAlarm											: ARRAY[1..20] OF INT;
	iActiveAlarms									: ARRAY[1..10] OF INT;								// 08/05/23 PS
	iActiveAlarmCount								: INT;												// 08/05/23 PS
	iCurrentAlarm									: INT;												// 08/05/23 PS
END_VAR

// Calvin - P_Alarm_Check
// Rev 1.00 - August 5, 2023

IF NOT gbAlarmsLoaded THEN
	A_LoadAlarms();
END_IF

IF tgb_Alarm_Reset THEN
	tgs_Alarm										:= '00';
	FOR i := 1 TO ALARM_COUNT DO
		gbAlarms[i]									:= FALSE;
	END_FOR
	tgb_Alarm_Reset									:= FALSE;
	eState											:= eIdle;
	tgi_Alarm_State									:= 0;
END_IF

// 08/05/23 PS - Updated to handle multiple alarms
IF giActiveAlarm > 0 THEN
	iActiveAlarmCount								:= SEL(iActiveAlarmCount < 10, iActiveAlarmCount, iActiveAlarmCount + 1);
	iActiveAlarms[iActiveAlarmCount]				:= giActiveAlarm;
	giActiveAlarm									:= 0;
END_IF

ftrigClearError(CLK:= tgb_Active_Alarm);
IF ftrigClearError.Q THEN
	FOR i:= 1 TO 9 DO
		iActiveAlarms[i] 							:= iActiveAlarms[i+1];
	END_FOR
	iActiveAlarms[10]								:= 0;
	iActiveAlarmCount								:= iActiveAlarmCount - 1;
END_IF

IF tonAlarmTimer.Q THEN
	IF iActiveAlarmCount > 0 THEN
		iCurrentAlarm								:= iActiveAlarms[1];
		tgb_Active_Alarm 							:= TRUE;
		gbAlarms[iCurrentAlarm]						:= TRUE;
		tgs_Active_Alarm							:= CONCAT(gsAlarms[iCurrentAlarm], gsTempAlarm);
		gsTempAlarm									:= '';
	END_IF
END_IF

rtrigCheckErrors(CLK:= tgb_Half_Sec_Pulse);
IF rtrigCheckErrors.Q THEN
	iErrorCount										:= 0;
	FOR i := 1 TO ALARM_COUNT DO
		IF gbAlarms[i] THEN
			iErrorCount								:= iErrorCount + 1;
			iAlarm[iErrorCount]						:= i;
		END_IF
	END_FOR
	iCount											:= iCount + 1;

	IF iErrorCount > 1 THEN
		IF iCount >= 1 AND iCount <= 3 THEN
			tgs_Alarm								:= gsAlarms[iAlarm[iDisplayAlarm]];
		ELSE
			tgs_Alarm								:= '00';							// Blank label for one half second
			iCount									:= 0;
			iDisplayAlarm							:= iDisplayAlarm + 1;
			IF iDisplayAlarm > iErrorCount THEN
				iDisplayAlarm 						:= 1;
			END_IF
		END_IF
	ELSIF iErrorCount = 1 THEN
		iCount										:= 0;
		iDisplayAlarm								:= 1;
		tgs_Alarm									:= gsAlarms[iAlarm[1]];
	ELSE
		iCount										:= 0;
		tgs_Alarm 									:= ALARM_00;
	END_IF
END_IF

tonAlarmTimer(IN:= NOT tgb_Active_Alarm, PT:= T#750MS);

IF tgb_File_Save_Error THEN
	tgb_File_Save_Error								:= FALSE;
	giActiveAlarm									:= eSystem_Alarm;
	gsAlarmInfo[eSystem_Alarm]						:= gsFileSaveError;
	gbAlarms[eSystem_Alarm]							:= TRUE;
	gbAlarmsLoaded									:= FALSE;                                                       // Clear flag to reload alarms with alarm string
END_IF

ACTION A_LoadAlarms:
// Calvin - P_Alarm_Check.A_LoadAlarms
// Rev 1.00 - June 12, 2023

gsAlarms[0]										:= ALARM_00;
gsAlarms[1]										:= CONCAT(ALARM_01, gsAlarmInfo[eWarmup_Alarm]);
gsAlarms[2]										:= CONCAT(ALARM_02, gsAlarmInfo[eEvacuation_Alarm]);
gsAlarms[3]										:= CONCAT(ALARM_03, gsAlarmInfo[eSteamBypass_Alarm]);
gsAlarms[4]										:= CONCAT(ALARM_04, gsAlarmInfo[eDesorption_Alarm]);
gsAlarms[5]										:= CONCAT(ALARM_05, gsAlarmInfo[eRepressurization_Alarm]);
gsAlarms[6]										:= CONCAT(ALARM_06, gsAlarmInfo[eAdsorption_Alarm]);
gsAlarms[7]										:= CONCAT(ALARM_07, gsAlarmInfo[eSystem_Alarm]);
gsAlarms[8]										:= CONCAT(ALARM_08, gsAlarmInfo[eTC_Alarm]);
gsAlarms[9]										:= CONCAT(ALARM_09, gsAlarmInfo[eSystem_Alarm]);
gsAlarms[10]									:= ALARM_10;
gsAlarms[11]									:= ALARM_11;
gsAlarms[12]									:= ALARM_12;
gsAlarms[13]									:= ALARM_13;
gsAlarms[14]									:= ALARM_14;
gsAlarms[15]									:= ALARM_15;
gsAlarms[16]									:= ALARM_16;
gsAlarms[17]									:= ALARM_17;
gsAlarms[18]									:= ALARM_18;
gsAlarms[19]									:= ALARM_19;
gsAlarms[20]									:= ALARM_20;
gsAlarms[21]									:= CONCAT(ALARM_21, gsAlarmInfo[21]);
gsAlarms[22]									:= CONCAT(ALARM_22, gsAlarmInfo[22]);
gsAlarms[23]									:= ALARM_23;
gsAlarms[24]									:= ALARM_24;
gsAlarms[25]									:= ALARM_25;
gsAlarms[26]									:= ALARM_26;
gsAlarms[27]									:= ALARM_27;
gsAlarms[28]									:= ALARM_28;
gsAlarms[29]									:= ALARM_29;
gsAlarms[30]									:= ALARM_30;
gsAlarms[31]									:= ALARM_31;
gsAlarms[32]									:= ALARM_32;
gsAlarms[33]									:= ALARM_33;
gsAlarms[34]									:= ALARM_34;
gsAlarms[35]									:= ALARM_35;
gsAlarms[36]									:= ALARM_36;
gsAlarms[37]									:= ALARM_37;
gsAlarms[38]									:= ALARM_38;
gsAlarms[39]									:= ALARM_39;
gsAlarms[40]									:= ALARM_40;
gsAlarms[41]									:= ALARM_41;
gsAlarms[42]									:= ALARM_42;
gsAlarms[43]									:= ALARM_43;
gsAlarms[44]									:= ALARM_44;
gsAlarms[45]									:= ALARM_45;
gsAlarms[46]									:= ALARM_46;
gsAlarms[47]									:= ALARM_47;
gsAlarms[48]									:= ALARM_48;
gsAlarms[49]									:= ALARM_49;
gbAlarmsLoaded									:= TRUE;
END_ACTION

END_PROGRAM

// ---- POUs/P_HeaterControl.TcPOU
PROGRAM P_HeaterControl
VAR
	TempControl_1									: FB_Temp_Control;
	TempControl_2									: FB_Temp_Control;
	TempControl_3									: FB_Temp_Control;
	TempControl_4									: FB_Temp_Control;
	TempControl_5									: FB_Temp_Control;
	TempControl_6									: FB_Temp_Control;
END_VAR

// Calvin - P_HeaterControl
// Rev 1.00 - May 20, 2023

IF giActiveAlarm <> 1 AND tgb_HT_1_On THEN
	TempControl_1(
		Set_Point									:= tgr_HT_1_SP, 
		Temperature									:= tgr_TI_1, 
		I_Range 									:= tgr_HT_I_Range, 
		Pid_Cycle_Time								:= PID_CYCLE_TIME, 
		Pid_Kp										:= tgr_HT_P_Value, 
		Pid_Tn										:= tgr_HT_I_Value, 
		Pid_Tv										:= 0, 
		Pid_Td										:= 0,
		Base_Output									:= tgr_HT_1_Base_Output,
		Manual_Output								:= tgr_HT_1_Manual_Output,
		Output										=> HT_1_CTRL);
ELSE
	HT_1_CTRL										:= 0;
	HT_1_RELAY										:= FALSE;
END_IF
		
IF giActiveAlarm <> 1 AND tgb_HT_2_On THEN
	TempControl_2(
		Set_Point									:= tgr_HT_2_SP, 
		Temperature									:= tgr_TI_2, 
		I_Range 									:= tgr_HT_I_Range,
		Pid_Cycle_Time								:= PID_CYCLE_TIME, 
		Pid_Kp										:= tgr_HT_P_Value, 
		Pid_Tn										:= tgr_HT_I_Value, 
		Pid_Tv										:= 0, 
		Pid_Td										:= 0, 
		Base_Output									:= tgr_HT_2_Base_Output,
		Manual_Output								:= tgr_HT_2_Manual_Output, 
		Output										=> HT_2_CTRL);
ELSE
	HT_2_CTRL										:= 0;
	HT_2_RELAY										:= FALSE;
END_IF
		
IF giActiveAlarm <> 1 AND tgb_HT_3_On THEN
	TempControl_3(
		Set_Point									:= tgr_HT_3_SP, 
		Temperature									:= tgr_TI_3, 
		I_Range 									:= tgr_HT_I_Range,
		Pid_Cycle_Time								:= PID_CYCLE_TIME, 
		Pid_Kp										:= tgr_HT_P_Value, 
		Pid_Tn										:= tgr_HT_I_Value, 
		Pid_Tv										:= 0, 
		Pid_Td										:= 0, 
		Base_Output									:= tgr_HT_3_Base_Output,
		Manual_Output								:= tgr_HT_3_Manual_Output, 
		Output										=> HT_3_CTRL);
ELSE                                				
	HT_3_CTRL										:= 0;
	HT_3_RELAY										:= FALSE;
END_IF
		
IF giActiveAlarm <> 1 AND tgb_HT_4_On THEN
	TempControl_4(
		Set_Point									:= tgr_HT_4_SP, 
		Temperature									:= tgr_TI_4, 
		I_Range 									:= tgr_HT_I_Range,
		Pid_Cycle_Time								:= PID_CYCLE_TIME, 
		Pid_Kp										:= tgr_HT_P_Value, 
		Pid_Tn										:= tgr_HT_I_Value, 
		Pid_Tv										:= 0, 
		Pid_Td										:= 0,
		Base_Output									:= tgr_HT_4_Base_Output,
		Manual_Output								:= tgr_HT_4_Manual_Output, 
		Output										=> HT_4_CTRL);
ELSE                            				
	HT_4_CTRL										:= 0;
	HT_4_RELAY										:= FALSE;
END_IF                          	
		
IF giActiveAlarm <> 1 AND tgb_HT_5_On THEN
	TempControl_5(
		Set_Point									:= tgr_HT_5_SP, 
		Temperature									:= tgr_TI_5, 
		I_Range 									:= tgr_HT_I_Range,
		Pid_Cycle_Time								:= PID_CYCLE_TIME, 
		Pid_Kp										:= tgr_HT_P_Value, 
		Pid_Tn										:= tgr_HT_I_Value, 
		Pid_Tv										:= 0, 
		Pid_Td										:= 0,
		Base_Output									:= tgr_HT_5_Base_Output,
		Manual_Output								:= tgr_HT_5_Manual_Output,
		Output										=> HT_5_CTRL);
ELSE                        				
	HT_5_CTRL										:= 0;
	HT_5_RELAY										:= FALSE;
END_IF
		
IF giActiveAlarm <> 1 AND tgb_HT_6_On THEN
	TempControl_6(
		Set_Point									:= tgr_HT_6_SP, 
		Temperature									:= tgr_TI_6, 
		I_Range 									:= tgr_HT_I_Range,
		Pid_Cycle_Time								:= PID_CYCLE_TIME, 
		Pid_Kp										:= tgr_HT_P_Value, 
		Pid_Tn										:= tgr_HT_I_Value, 
		Pid_Tv										:= 0, 
		Pid_Td										:= 0, 
		Base_Output									:= tgr_HT_6_Base_Output,
		Manual_Output								:= tgr_HT_6_Manual_Output,
		Output										=> HT_6_CTRL);
ELSE                                	
	HT_6_CTRL							:= 0;
	HT_6_RELAY							:= FALSE;
END_IF                              	
	
tgr_HT_1_Ctrl						:= INT_TO_REAL(HT_1_CTRL);
tgr_HT_2_Ctrl						:= INT_TO_REAL(HT_2_CTRL);
tgr_HT_3_Ctrl						:= INT_TO_REAL(HT_3_CTRL);
tgr_HT_4_Ctrl						:= INT_TO_REAL(HT_4_CTRL);
tgr_HT_5_Ctrl						:= INT_TO_REAL(HT_5_CTRL);
tgr_HT_6_Ctrl						:= INT_TO_REAL(HT_6_CTRL);

END_PROGRAM

// ---- POUs/Function_Blocks/FB_Temp_Control.TcPOU
FUNCTION_BLOCK FB_Temp_Control
VAR_INPUT
	Set_Point										: REAL;				// Control set point
	Temperature										: REAL;				// Current control loop temperature
	I_Range											: REAL;				// Range that Integral value is active
	Pid_Cycle_Time									: REAL;				// PID cycle time - matches task time
	Pid_Kp											: REAL;				// Proportional gain
	Pid_Tn											: REAL;				// Integral gain
	Pid_Tv											: REAL;				// Derivative gain
	Pid_Td											: REAL;				// Derivative damping time
	Base_Output										: REAL;				// Estimated output value to hold setpoint
	Base_I_Factor									: REAL;				// Base Integral gain
	Base_I_Time										: REAL;				// Base Integral time
	Manual_Output									: REAL;				// Manual heater output
	Maximum_Output									: REAL := 32767;	// Maximum output value allowed 
END_VAR
VAR_OUTPUT
	Output											: INT;				// Integer output to control PWM for heater relay
	Current_Base									: REAL;
END_VAR
VAR
	bReset											: BOOL;				// Reset PID FB on set point change
	rOut											: REAL;				// Calculated output
	rSetPoint										: REAL := 0;		// Last set point - reset on change
	rBase											: REAL;
	rBaseTn											: REAL;
	rError											: REAL;										
	lrTn											: LREAL;			// Integral gain calculation
	lrOut											: LREAL;			// PID FB output
	fb_BasicPID										: FB_BasicPID;
	tonBase											: TON;
END_VAR

// FB_Temp_Control
// Rev 1.00 - May 10, 2023

IF Set_Point <> rSetPoint THEN																									// Check if set point has changed
	bReset											:= TRUE;																	// Reset function block if it has changed
	rSetPoint 										:= Set_Point;																// Save new value to reset check
	rBase											:= Base_Output;
ELSE
	bReset											:= FALSE;																	// No change, do not reset
END_IF

// Control heater output & PID loop based on current temperature and the set point range
rError												:= Set_Point - Temperature;
IF ABS(rError) <= I_Range THEN
	lrTn											:= REAL_TO_LREAL(Pid_Tn);													// Use Integral gain only if within range (Proportional + base otherwise)
	rBaseTn											:= Base_I_Factor;
ELSE
	lrTn											:= 0;
	rBaseTn											:= 0;
END_IF

IF tgb_Manual_Heater_Mode THEN
	rOut											:= REAL_TO_INT(Manual_Output);
ELSE
	fb_BasicPID(
		fSetpointValue								:= Set_Point,
		fActualValue								:= Temperature,
		bReset										:= bReset,
		fCtrlCycleTime								:= Pid_Cycle_Time,
		fKp											:= Pid_Kp,
		fTn											:= lrTn,
		fTv											:= REAL_TO_LREAL(Pid_Tv),
		fTd											:= REAL_TO_LREAL(Pid_Td),
		fCtrlOutput									=> lrOut,
		nErrorStatus								=> );

	IF tonBase.Q THEN
		tonBase(IN:= FALSE);
		rBase										:= rBase + rError * Base_I_Factor; 
	END_IF
	
	rOut											:= LREAL_TO_REAL(lrOut) + rBase;
	rOut											:= SEL(rOut < 0, SEL(rOut > Maximum_Output, rOut, Maximum_Output), 0);		// Keep PID output within range of INT value
END_IF

Output												:= REAL_TO_INT(rOut);
tonBase(IN:= TRUE, PT:= REAL_TO_TIME(Base_I_Time));

END_FUNCTION_BLOCK

// ---- POUs/P_VFD_Test.TcPOU
PROGRAM P_VFD_Test
VAR
	tonVFDTest					: TON;
	ftrigStop					: F_TRIG;
END_VAR

// Calvin - P_VFD_Test
// Rev 1.00 - July 14, 2023

IF gbVFDTest THEN
	tgr_IP_1102A								:= 100;
	tgr_IP_1102B								:= 100;
	IF tgb_IP_1102A_Open AND tgb_IP_1102B_Open AND tonVFDTest.Q THEN
		tonVFDTest(IN:= FALSE);
		IF tgr_HS_1102 = 80 THEN
			tgr_HS_1102							:= 0;
		ELSE
			tgr_HS_1102							:= 80;
		END_IF
	END_IF
	tonVFDTest(IN:= TRUE, PT:= T#30S);
END_IF

ftrigStop(CLK:= gbVFDTest);
IF ftrigStop.Q THEN
	tgr_HS_1102									:= 0;
	tgr_IP_1102A								:= 0;
	tgr_IP_1102B								:= 0;
END_IF

END_PROGRAM
